(* CODESYS project OC_EtherCAT.library
   DefaultNamespace: OC_EtherCAT
   Description: Open Commissioning TwinCAT EtherCAT Library
   Author: SpiraTec AG
   Title: OC_EtherCAT
   Version: 1.1.8
   Company: Open Commissioning
   Placeholder: OC_EtherCAT

Project tree, tasks and I/O mapping:
  libraries: OC_Core, 1.3.1 (Open Commissioning); OC_TwinSAFE, 1.0.2 (Open Commissioning); Tc2_Math, 3.4.4.0 (Beckhoff Automation GmbH); Tc2_Standard, 3.4.5.0 (Beckhoff Automation GmbH); Tc2_System, 3.6.4.0 (Beckhoff Automation GmbH); Tc3_Module, 3.4.5.0 (Beckhoff Automation GmbH); TcUnit, 1.3.0.0 (www.tcunit.org)
  Devices/
    Drives/
      DS402/
        data type E_DS402_State
        function block FB_DS402_CSP [ST]: Cycle, eState, fbEncoder, GetControlData, InitRun, SetStatusData
        function block FB_DS402_FSM [ST]: bError, eState, IsDisableOperation, IsDisableVoltage, IsEnableOperation, IsFaultReset, IsQuickStop, IsShutdown, IsSwitchOn, nControl, nStatus, ResetError, S0_NotReadyToSwitchOn, S1_SwitchOnDisabled, S2_ReadyToSwitchOn, S3_SwitchedOn, S4_OperationEnabled, S5_Fault, S6_FaultReactionActive, S7_QuickStopActive
        data type ST_DS402_ControlWord
        data type ST_DS402_CSP_Config
        data type ST_DS402_CSP_Control
        data type ST_DS402_CSP_Status
        data type ST_DS402_StatusWord
      Mitsubishi/
        function block FB_Mitsubishi_MRJ4TM [ST]: Cycle, eState, fbEncoder, GetControlData, InitRun, SetStatusData
        data type ST_Mitsubishi_MRJ4TM_Config
        data type ST_Mitsubishi_MRJ4TM_Control
        data type ST_Mitsubishi_MRJ4TM_Status
      Sercos/
        data type E_Sercos_State
        function block FB_Sercos_FSM [ST]: bError, eState, nControl, nStatus, S1_NotReadyToSwitchOn, S2_SwitchOnDisabled, S3_ReadyToSwitchOn, S4_SwitchOn, S5a_DriveInOperation, S5b_Halt, S6_QuickStop, S7_FaultReactionActive, S8_Fault
        function block FB_Sercos_VC [ST]: Cycle, eState, fbEncoder, GetControlData, GetTargetVelocity, InitRun, Motion, SetStatusData
        data type ST_Sercos_ControlWord
        data type ST_Sercos_StatusWord
        data type ST_Sercos_VC
        data type ST_Sercos_VC_Config
        data type ST_Sercos_VC_Control
        data type ST_Sercos_VC_Status
    Terminals/
      FB_Beckhoff_EL6001/
        data type E_Beckhoff_EL6001_State
        function block FB_Beckhoff_EL6001 [ST]: BufferFull, Control, FramingError, InitAccepted, InitRequest, OverrunError, ParityError, ReceiveAccepted, ReceiveRequest, SendContinuous, State, TransmitAccepted, TransmitRequest
      function block FB_Beckhoff_EJ1918 [ST]: FB_init
      function block FB_Beckhoff_EK1914 [ST]: FB_init
      function block FB_Beckhoff_EL1904 [ST]: FB_init
      function block FB_Beckhoff_EL1918 [ST]: FB_init
      function block FB_Beckhoff_EL2904 [ST]: FB_init
      function block FB_Beckhoff_EL5152 [ST]: Control1, Control2, Counter1, Counter2, Period1, Period2, SetCounter1, SetCounter2, Status1, Status2
      function block FB_FSOE_19 [ST]: FB_init
      data type ST_Baumer_Encoder
      data type ST_Beckhoff_16DI
      data type ST_Beckhoff_16DO
      data type ST_Beckhoff_2AI
      data type ST_Beckhoff_4AI
      data type ST_Beckhoff_4AO
      data type ST_Beckhoff_4DI
      data type ST_Beckhoff_4DI_4DO
      data type ST_Beckhoff_4DO
      data type ST_Beckhoff_8DI
      data type ST_Beckhoff_8DI_8DO
      data type ST_Beckhoff_8DO
      data type ST_Beckhoff_EL3403
      data type ST_Beckhoff_EL5002
      data type ST_Beckhoff_EL9110
      data type ST_Beckhoff_EL9410
      data type ST_CoE402
      data type ST_Gefran_GFX4
      data type ST_Mitsubishi_MRJ4TM
      data type ST_SEW_SimMovitrac
*)

// Devices/Drives/DS402/E_DS402_State
{attribute 'qualified_only'}
{attribute 'strict'}
{attribute 'conditionalshow'}
TYPE E_DS402_State :
(
	S0_NotReadyToSwitchOn,
	S1_SwitchOnDisabled,
	S2_ReadyToSwitchOn,
	S3_SwitchedOn,
	S4_OperationEnabled,
	S5_Fault,
	S6_FaultReactionActive,
	S7_QuickStopActive
);
END_TYPE

// Devices/Drives/DS402/ST_DS402_ControlWord
(*
	Object 6040h: Control word (DS402)	
*)
{attribute 'pack_mode' := '0'}
TYPE ST_DS402_ControlWord :
STRUCT
	b0_SwitchOn 					: BIT;
	b1_EnableVoltage				: BIT;
	b2_QuickStop					: BIT;
	b3_EnableOperation				: BIT;
	b4_OperationModeSpecific		: BIT;
	b5_OperationModeSpecific		: BIT;
	b6_OperationModeSpecific		: BIT;
	b7_FaultReset					: BIT;
	b8_Reserved						: BIT;
	b9_Reserved						: BIT;
	b10_Reserved					: BIT;
	b11_Reserved					: BIT;
	b12_Reserved					: BIT;
	b13_Reserved					: BIT;
	b14_Reserved					: BIT;
	b15_Reserved					: BIT;
END_STRUCT
END_TYPE

// Devices/Drives/DS402/ST_DS402_CSP_Config
{attribute 'pack_mode' := '0'}
TYPE ST_DS402_CSP_Config :
STRUCT	
	bForceMode			: BOOL; //Ignore process data from fieldbus.	
	bSwapProcessData	: BOOL; //Reverse process data byte order from/to fieldbus.
	fPositionOffset		: LREAL := 0.0;	
	bSyncOpMode			: BOOL := TRUE;
END_STRUCT
END_TYPE

// Devices/Drives/DS402/ST_DS402_CSP_Control
(*
	Control struct for Cyclic synchronous position mode(CSP)
	0x1600 (DS402 Controlword)
	0x1606 (DS402 Target position)
*)
{attribute 'pack_mode' := '0'}
TYPE ST_DS402_CSP_Control :
STRUCT
	nControlWord 		: ST_DS402_ControlWord; //0x1600 (DS402 Controlword)
	nTargetPosition		: DINT;	//DS402 Target position [INC]	
END_STRUCT
END_TYPE

// Devices/Drives/DS402/ST_DS402_CSP_Status
(*
	Status struct for Cyclic synchronous position mode(CSP)
	0x1A00 (DS402 Statusword)
	0x1A01 (DS402 Position actual value)
	0x1A04 (DS402 Following error actual value)
*)
{attribute 'pack_mode' := '0'}
TYPE ST_DS402_CSP_Status :
STRUCT
	nStatusWord 		: ST_DS402_StatusWord; //0x1A00 (DS402 Statusword)
	nActualPosition		: DINT;	//0x1A01 (DS402 Position actual value) [INC]
	nErrorPosition		: DINT;	//0x1A04 (DS402 Following error actual value) [INC]	
END_STRUCT
END_TYPE

// Devices/Drives/DS402/ST_DS402_StatusWord
(*
	Object 6041h: Status word (DS402)
*)
{attribute 'pack_mode' := '0'}
TYPE ST_DS402_StatusWord :
STRUCT
	b0_ReadyToSwitchOn 				: BIT; 
	b1_SwitchedOn 					: BIT; 
	b2_OperationEnabled 			: BIT; 
	b3_Fault						: BIT; 
	b4_VoltageEnabled				: BIT; 
	b5_QuickStop					: BIT;
	b6_SwitchOnDisabled				: BIT; 
	b7_Warning						: BIT; 
	b8_Synchranisation				: BIT; 
	b9_Remote						: BIT;
	b10_TargetReached				: BIT;
	b11_InternalLimitActive			: BIT; 
	b12_OperationModeSpecific		: BIT; 
	b13_OperationModeSpecific		: BIT; 
	b14_OperationModeSpecific		: BIT; 
	b15_ClosedLoopActive			: BIT;
END_STRUCT
END_TYPE

// Devices/Drives/Mitsubishi/ST_Mitsubishi_MRJ4TM_Config
{attribute 'pack_mode' := '0'}
TYPE ST_Mitsubishi_MRJ4TM_Config :
STRUCT	
	bForceMode			: BOOL; //Ignore process data from fieldbus.	
	bSwapProcessData	: BOOL; //Reverse process data byte order from/to fieldbus.
	fPositionOffset		: LREAL := 0.0;	
	bSyncOpMode			: BOOL := TRUE;
END_STRUCT
END_TYPE

// Devices/Drives/Mitsubishi/ST_Mitsubishi_MRJ4TM_Control
(*
	
*)
{attribute 'pack_mode' := '0'}
TYPE ST_Mitsubishi_MRJ4TM_Control :
STRUCT
	nModesOfOperation 				: SINT;
	nControlWord 					: ST_DS402_ControlWord; //0x1600 (DS402 Controlword)
	nControlID1						: UINT;
	nControlID2						: UINT;
	nControlID3						: UINT;
	nTargetPosit					: DINT;
	nTargetVeloc					: DINT;
	nVelocityLimitValue				: UDINT;
	nTargetTorque					: INT;
	nPositiveTorqueLimitValue		: UINT;
	nNegativeTorqueLimitValue 		: UINT;
	nTouchProbeFunction				: UINT;
END_STRUCT
END_TYPE

// Devices/Drives/Mitsubishi/ST_Mitsubishi_MRJ4TM_Status
(*
	
*)
{attribute 'pack_mode' := '0'}
TYPE ST_Mitsubishi_MRJ4TM_Status :
STRUCT
	nModesOfOperationDisplay 		: SINT;
	nStatusWord 					: ST_DS402_StatusWord; //0x1A00 (DS402 Statusword)
	nStatusDO1						: UINT;
	nStatusDO2						: UINT;
	nStatusDO3						: UINT;
	nPositionActualValue			: DINT;
	nVelocityActualValue			: DINT;
	nFollowingErrorActualValue		: DINT;
	nTorqueActualValue				: INT;
	nTouchProbeStatus				: UINT;
	nTouchProbePos1PosValue			: DINT;
	nTouchProbePos1NegValue			: DINT;
	nTouchProbePos2PosValue			: DINT;
	nTouchProbePos2NegValue			: DINT;
END_STRUCT
END_TYPE

// Devices/Drives/Sercos/E_Sercos_State
{attribute 'qualified_only'}
{attribute 'strict'}
{attribute 'conditionalshow'}
TYPE E_Sercos_State :
(
	S1_NotReadyToSwitchOn,
	S2_SwitchOnDisabled,
	S3_ReadyToSwitchOn,
	S4_SwitchOn,
	S5a_DriveInOperation,
	S5b_Halt,
	S6_QuickStop,
	S7_FaultReactionActive,
	S8_Fault
);
END_TYPE

// Devices/Drives/Sercos/ST_Sercos_ControlWord
(*
	S-0-0134 Drive Control
	https://product-help.schneider-electric.com/Machine%20Expert/V1.2/en/ATV340SUG/ATV340SUG/STI_Software_Setup/STI_Software_Setup-21.htm#XREF_D_SE_0083221_1
*)
{attribute 'pack_mode' := '1'}
TYPE ST_Sercos_ControlWord :
STRUCT
	b0_Reserved 					: BIT;
	b1_Reserved						: BIT;
	b2_Reserved						: BIT;
	b3_Reserved						: BIT;
	b4_Reserved						: BIT;
	b5_Reserved						: BIT;
	b6_Reserved						: BIT;
	b7_Reserved						: BIT;
	b8_Reserved						: BIT; //Reserved (=0)
	b9_Reserved						: BIT; //Reserved (=0)
	b10_OperationMode				: BIT; //0 = Primary operation mode
	b11_Reserved					: BIT;
	b12_Reserved					: BIT; 
	b13_Halt						: BIT; //Drive halt, 1 --> 0 = halt, 0 --> 1 = restart
	b14_Start						: BIT; //Drive start, 1 --> 0 = Stop, 0 -> 1 = Start 
	b15_Enable						: BIT; //Drive enable, 1 --> 0 = drive disabled, 0 -> 1 = drive enabled
END_STRUCT
END_TYPE

// Devices/Drives/Sercos/ST_Sercos_StatusWord
(*
	S-0-0135 Drive Status
	https://product-help.schneider-electric.com/Machine%20Expert/V1.2/en/ATV340SUG/ATV340SUG/STI_Software_Setup/STI_Software_Setup-22.htm#XREF_D_SE_0083227_1
*)
{attribute 'pack_mode' := '1'}
TYPE ST_Sercos_StatusWord :
STRUCT
	b0_Reserved 					: BIT;
	b1_Reserved						: BIT;
	b2_Reserved						: BIT;
	b3_CommandProcessing			: BIT; //Status command value processing if 0 = ignored
	b4_Halt							: BIT; //Drive halt, 0 = inactive, 1 = active
	b5_PositionFeedback				: BIT; //Position feedback value status (S-0-0403)
	b6_Reserved						: BIT;
	b7_QuickStop					: BIT; //Quick stop, 0 = inactive, 1 = active
	b8_Reserved						: BIT; //Reserved (=0)
	b9_Reserved						: BIT; //Reserved (=0)
	b10_OperationMode				: BIT; //0 = Primary operation mode
	b11_Reserved					: BIT;
	b12_Warning						: BIT; //Warning, 0 = No warning, 1 = Warning
	b13_Error						: BIT; //Drive shut-down error, 0 = No error, 1 = Error
	b14_ReadyToOperate				: BIT; //00 = Not ready to switch on, 01 = Switch on disabled, main power disabled
	b15_ReadyToOperate				: BIT; //10 = Switch on, 11 = Drive enabled
END_STRUCT
END_TYPE

// Devices/Drives/Sercos/ST_Sercos_VC
{attribute 'pack_mode' := '1'} 
TYPE ST_Sercos_VC :
STRUCT
	stControl		AT %I* : ST_Sercos_VC_Control;
	stStatus		AT %Q* : ST_Sercos_VC_Status;
END_STRUCT
END_TYPE

// Devices/Drives/Sercos/ST_Sercos_VC_Config
{attribute 'pack_mode' := '0'}
TYPE ST_Sercos_VC_Config :
STRUCT	
	bForceMode				: BOOL; //Ignore process data from fieldbus.	
	bSwapProcessData		: BOOL; //Reverse process data byte order from/to fieldbus.	
	bIsLinkOutputVelocity	: BOOL; //If TRUE, link output is velocity value
	fReferenceVelocity 		: REAL := 1000.0;
	fNormalizationFactor	: REAL := 80000;
END_STRUCT
END_TYPE

// Devices/Drives/Sercos/ST_Sercos_VC_Control
(*
	Sercos Velocity Control
	MDT: S-0-0134 Master control word
	MDT: S-0-0036 Velocity command value
*)
{attribute 'pack_mode' := '0'}
TYPE ST_Sercos_VC_Control :
STRUCT
	nControlWord 			: ST_Sercos_ControlWord; //S-0-0134 Master control word
	nVelocityCommand		: DINT;	//S-0-0036 Velocity command value
END_STRUCT
END_TYPE

// Devices/Drives/Sercos/ST_Sercos_VC_Status
(*
	Sercos Velocity Control
	AT: S-0-0135 Drive Status word
	AT: S-0-0051 Position feedback 1 value
*)
{attribute 'pack_mode' := '0'}
TYPE ST_Sercos_VC_Status :
STRUCT
	nStatusWord 			: ST_Sercos_StatusWord; //S-0-0135 Drive Status word
	nPositionFeedback		: DINT;	//S-0-0051 Position feedback 1 value
END_STRUCT
END_TYPE

// Devices/Terminals/FB_Beckhoff_EL6001/E_Beckhoff_EL6001_State
{attribute 'qualified_only'}
{attribute 'strict'}
TYPE E_Beckhoff_EL6001_State :
(
	INIT,
	READY,
	TRANSMIT, 
	RECEIVE
);
END_TYPE

// Devices/Terminals/ST_Baumer_Encoder
{attribute 'pack_mode' := '1'}
TYPE ST_Baumer_Encoder :
STRUCT
	nPosition		AT %Q*	:	UDINT;
	nWarnings		AT %Q*	:	UINT;
	nSystemTime		AT %Q*	:	UDINT; 
END_STRUCT
END_TYPE

// Devices/Terminals/ST_Beckhoff_16DI
{attribute 'pack_mode' := '1'} 
TYPE ST_Beckhoff_16DI :
STRUCT
	bIn1	AT %Q* : BIT;
	bIn2	AT %Q* : BIT;
	bIn3	AT %Q* : BIT;
	bIn4	AT %Q* : BIT;
	bIn5	AT %Q* : BIT;
	bIn6	AT %Q* : BIT;
	bIn7	AT %Q* : BIT;
	bIn8	AT %Q* : BIT;
	bIn9	AT %Q* : BIT;
	bIn10	AT %Q* : BIT;
	bIn11	AT %Q* : BIT;
	bIn12	AT %Q* : BIT;
	bIn13	AT %Q* : BIT;
	bIn14	AT %Q* : BIT;
	bIn15	AT %Q* : BIT;
	bIn16	AT %Q* : BIT;
END_STRUCT
END_TYPE

// Devices/Terminals/ST_Beckhoff_16DO
{attribute 'pack_mode' := '1'} 
TYPE ST_Beckhoff_16DO :
STRUCT
	bOut1	AT %I* : BIT;
	bOut2	AT %I* : BIT;
	bOut3	AT %I* : BIT;
	bOut4	AT %I* : BIT;
	bOut5	AT %I* : BIT;
	bOut6	AT %I* : BIT;
	bOut7	AT %I* : BIT;
	bOut8	AT %I* : BIT;
	bOut9	AT %I* : BIT;
	bOut10	AT %I* : BIT;
	bOut11	AT %I* : BIT;
	bOut12	AT %I* : BIT;
	bOut13	AT %I* : BIT;
	bOut14	AT %I* : BIT;
	bOut15	AT %I* : BIT;
	bOut16	AT %I* : BIT;
END_STRUCT
END_TYPE

// Devices/Terminals/ST_Beckhoff_2AI
{attribute 'pack_mode' := '1'} 
TYPE ST_Beckhoff_2AI :
STRUCT
	nStatus1	AT %Q* : UINT;
	nValue1		AT %Q* : INT;
	nStatus2	AT %Q* : UINT;
	nValue2		AT %Q* : INT;
	nStatus3	AT %Q* : UINT;
	nValue3		AT %Q* : INT;
	nStatus4	AT %Q* : UINT;
	nValue4		AT %Q* : INT;
END_STRUCT
END_TYPE

// Devices/Terminals/ST_Beckhoff_4AI
{attribute 'pack_mode' := '1'} 
TYPE ST_Beckhoff_4AI :
STRUCT
	nStatus1	AT %Q* : UINT;
	nValue1		AT %Q* : INT;
	nStatus2	AT %Q* : UINT;
	nValue2		AT %Q* : INT;
END_STRUCT
END_TYPE

// Devices/Terminals/ST_Beckhoff_4AO
{attribute 'pack_mode' := '1'} 
TYPE ST_Beckhoff_4AO :
STRUCT
	nAnalogOut1	AT %I* : UINT;
	nAnalogOut2	AT %I* : UINT;
	nAnalogOut3	AT %I* : UINT;
	nAnalogOut4	AT %I* : UINT;
END_STRUCT
END_TYPE

// Devices/Terminals/ST_Beckhoff_4DI
{attribute 'pack_mode' := '1'} 
TYPE ST_Beckhoff_4DI :
STRUCT
	bIn1	AT %Q* : BIT;
	bIn2	AT %Q* : BIT;
	bIn3	AT %Q* : BIT;
	bIn4	AT %Q* : BIT;	
END_STRUCT
END_TYPE

// Devices/Terminals/ST_Beckhoff_4DI_4DO
{attribute 'pack_mode' := '1'} 
TYPE ST_Beckhoff_4DI_4DO :
STRUCT
	bIn1	AT %Q* : BIT;
	bIn2	AT %Q* : BIT;
	bIn3	AT %Q* : BIT;
	bIn4	AT %Q* : BIT;	
	bOut1	AT %I* : BIT;
	bOut2	AT %I* : BIT;
	bOut3	AT %I* : BIT;
	bOut4	AT %I* : BIT;	
END_STRUCT
END_TYPE

// Devices/Terminals/ST_Beckhoff_4DO
{attribute 'pack_mode' := '1'} 
TYPE ST_Beckhoff_4DO :
STRUCT
	bOut1	AT %I* : BIT;
	bOut2	AT %I* : BIT;
	bOut3	AT %I* : BIT;
	bOut4	AT %I* : BIT;	
END_STRUCT
END_TYPE

// Devices/Terminals/ST_Beckhoff_8DI
{attribute 'pack_mode' := '1'} 
TYPE ST_Beckhoff_8DI :
STRUCT
	bIn1	AT %Q* : BIT;
	bIn2	AT %Q* : BIT;
	bIn3	AT %Q* : BIT;
	bIn4	AT %Q* : BIT;
	bIn5	AT %Q* : BIT;
	bIn6	AT %Q* : BIT;
	bIn7	AT %Q* : BIT;
	bIn8	AT %Q* : BIT;
END_STRUCT
END_TYPE

// Devices/Terminals/ST_Beckhoff_8DI_8DO
{attribute 'pack_mode' := '1'} 
TYPE ST_Beckhoff_8DI_8DO :
STRUCT
	bIn1	AT %Q* : BIT;
	bIn2	AT %Q* : BIT;
	bIn3	AT %Q* : BIT;
	bIn4	AT %Q* : BIT;
	bIn5	AT %Q* : BIT;
	bIn6	AT %Q* : BIT;
	bIn7	AT %Q* : BIT;
	bIn8	AT %Q* : BIT;
	bOut1	AT %I* : BIT;
	bOut2	AT %I* : BIT;
	bOut3	AT %I* : BIT;
	bOut4	AT %I* : BIT;
	bOut5	AT %I* : BIT;
	bOut6	AT %I* : BIT;
	bOut7	AT %I* : BIT;
	bOut8	AT %I* : BIT;
END_STRUCT
END_TYPE

// Devices/Terminals/ST_Beckhoff_8DO
{attribute 'pack_mode' := '1'} 
TYPE ST_Beckhoff_8DO :
STRUCT
	bOut1	AT %I* : BIT;
	bOut2	AT %I* : BIT;
	bOut3	AT %I* : BIT;
	bOut4	AT %I* : BIT;
	bOut5	AT %I* : BIT;
	bOut6	AT %I* : BIT;
	bOut7	AT %I* : BIT;
	bOut8	AT %I* : BIT;
END_STRUCT
END_TYPE

// Devices/Terminals/ST_Beckhoff_EL3403
TYPE ST_Beckhoff_EL3403 :
STRUCT
	nCurrent1		AT %Q* : UINT;
	nVoltage1		AT %Q* : UINT;
	nActivePower1	AT %Q* : UINT;
	nCurrent2		AT %Q* : UINT;
	nVoltage2		AT %Q* : UINT;
	nActivePower2	AT %Q* : UINT;	
	nCurrent3		AT %Q* : UINT;
	nVoltage3		AT %Q* : UINT;
	nActivePower3	AT %Q* : UINT;
END_STRUCT
END_TYPE

// Devices/Terminals/ST_Beckhoff_EL5002
TYPE ST_Beckhoff_EL5002 :
STRUCT
	nStatus1	AT %Q* : UINT;
	nCounter1	AT %Q* : UDINT;	
	nStatus2	AT %Q* : UINT;
	nCounter2	AT %Q* : UDINT;	
END_STRUCT
END_TYPE

// Devices/Terminals/ST_Beckhoff_EL9110
{attribute 'pack_mode' := '1'} 
TYPE ST_Beckhoff_EL9110 :
STRUCT
	bPowerOk	AT %Q* : BIT := TRUE;
END_STRUCT
END_TYPE

// Devices/Terminals/ST_Beckhoff_EL9410
{attribute 'pack_mode' := '1'} 
TYPE ST_Beckhoff_EL9410 :
STRUCT
	bUsUndervoltage	AT %Q* : BIT;
	bUpUndervoltage	AT %Q* : BIT;
END_STRUCT
END_TYPE

// Devices/Terminals/ST_CoE402
{attribute 'pack_mode' := '1'} 
TYPE ST_CoE402 :
STRUCT
	nControlWord	AT %I* : UINT;
	nTargetValue	AT %I* : DINT;
	nStatusWord		AT %Q* : UINT;
	nActualValue	AT %Q* : DINT;
END_STRUCT
END_TYPE

// Devices/Terminals/ST_Gefran_GFX4
{attribute 'pack_mode' := '1'} 
TYPE ST_Gefran_GFX4 :
STRUCT
	nProcessVariable1	AT %Q* : INT;
	nControllerStatus1	AT %Q* : UINT;	
	nOutputPower1		AT %Q* : INT;
	nProcessVariable2	AT %Q* : INT;
	nControllerStatus2	AT %Q* : UINT;	
	nOutputPower2		AT %Q* : INT;
	nProcessVariable3	AT %Q* : INT;
	nControllerStatus3	AT %Q* : UINT;	
	nOutputPower3		AT %Q* : INT;
	nProcessVariable4	AT %Q* : INT;
	nControllerStatus4	AT %Q* : UINT;	
	nOutputPower4		AT %Q* : INT;
	nLocalSetpoint1		AT %I* : INT;
	nLocalSetpoint2		AT %I* : INT;
	nLocalSetpoint3		AT %I* : INT;
	nLocalSetpoint4		AT %I* : INT;
END_STRUCT
END_TYPE

// Devices/Terminals/ST_Mitsubishi_MRJ4TM
{attribute 'pack_mode' := '1'} 
TYPE ST_Mitsubishi_MRJ4TM :
STRUCT
	nModesOfOperation 				AT %I* : SINT;
	nControlWord					AT %I* : UINT;
	nControlID1						AT %I* : UINT;
	nControlID2						AT %I* : UINT;
	nControlID3						AT %I* : UINT;
	nTargetPosit					AT %I* : DINT;
	nTargetVeloc					AT %I* : DINT;
	nVelocityLimitValue				AT %I* : UDINT;
	nTargetTorque					AT %I* : INT;
	nPositiveTorqueLimitValue		AT %I* : UINT;
	nNegativeTorqueLimitValue 		AT %I* : UINT;
	nTouchProbeFunction				AT %I* : UINT;
	
	nModesOfOperationDisplay 		AT %Q* : SINT;
	nStatusWord						AT %Q* : UINT;
	nStatusDO1						AT %Q* : UINT;
	nStatusDO2						AT %Q* : UINT;
	nStatusDO3						AT %Q* : UINT;
	nPositionActualValue			AT %Q* : DINT;
	nVelocityActualValue			AT %Q* : DINT;
	nFollowingErrorActualValue		AT %Q* : DINT;
	nTorqueActualValue				AT %Q* : INT;
	nTouchProbeStatus				AT %Q* : UINT;
	nTouchProbePos1PosValue			AT %Q* : DINT;
	nTouchProbePos1NegValue			AT %Q* : DINT;
	nTouchProbePos2PosValue			AT %Q* : DINT;
	nTouchProbePos2NegValue			AT %Q* : DINT;
END_STRUCT
END_TYPE

// Devices/Terminals/ST_SEW_SimMovitrac
{attribute 'pack_mode' := '1'}
TYPE ST_SEW_SimMovitrac :
STRUCT
	PI1		AT %Q* : WORD;
	PI2		AT %Q* : WORD;
	PI3		AT %Q* : WORD;
	PO1		AT %I* : WORD;
	PO2		AT %I* : WORD;
	PO3		AT %I* : WORD;
END_STRUCT
END_TYPE

// Devices/Drives/DS402/FB_DS402_CSP
(*
	DS402 with Cyclic synchronous position mode(CSP)
	SM2 PDO: 0x1600 (DS402 Controlword)	
	SM2 PDO: 0x1606 (DS402 Target position)
	SM3 PDO: 0x1A00 (DS402 Statusword)	
	SM3 PDO: 0x1A01 (DS402 Position actual value)
	SM3 PDO: 0x1A04 (DS402 Following error actual value)
*)
{attribute 'reflection'} 
FUNCTION_BLOCK FB_DS402_CSP EXTENDS FB_LinkDataReal 
VAR_INPUT
	pControl			: PVOID; //Pocess data from fieldbus, 6 BYTES FROM FIELDBUS
	pStatus				: PVOID; //Pocess data to fieldbus, 6 BYTES FROM FIELDBUS		
	stControl	 		: ST_DS402_CSP_Control;
	stConfig			: ST_DS402_CSP_Config;
	bSTO 				: BOOL := TRUE;
END_VAR

VAR_OUTPUT
	stStatus 			: ST_DS402_CSP_Status;	
END_VAR

VAR		
	{attribute 'instance-path'} 
    {attribute 'noinit'} 
    _sPath 				: STRING;
	_fbStateMachine 	: FB_DS402_FSM;
	_fbEncoder 			: FB_Encoder;	
END_VAR

SUPER^();
InitRun();

GetControlData();
Cycle();
SetStatusData();

METHOD PRIVATE Cycle
IF NOT bSTO THEN RETURN; END_IF

_fbStateMachine.stControl := stControl.nControlWord;
_fbStateMachine();
stStatus.nStatusWord := _fbStateMachine.stStatus;

IF (_fbStateMachine._eState = E_DS402_State.S4_OperationEnabled) THEN	
	
	_fbEncoder.fValue :=  stConfig.fPositionOffset + _fbEncoder.INC_TO_LREAL(stControl.nTargetPosition, 1);
	_fbEncoder();
END_IF

IF stConfig.bSyncOpMode THEN
	stStatus.nStatusWord.b12_OperationModeSpecific := stControl.nControlWord.b4_OperationModeSpecific;
	stStatus.nStatusWord.b13_OperationModeSpecific := stControl.nControlWord.b5_OperationModeSpecific;
	stStatus.nStatusWord.b14_OperationModeSpecific := stControl.nControlWord.b6_OperationModeSpecific;
END_IF


stStatus.nActualPosition := _fbEncoder.nResult;

//Set Link Data
ControlData := LREAL_TO_REAL(_fbEncoder.fResult);
END_METHOD

PROPERTY eState : E_DS402_State
GET
eState := _fbStateMachine.eState;
END_GET
END_PROPERTY

PROPERTY PUBLIC fbEncoder : REFERENCE TO FB_Encoder
GET
fbEncoder REF= _fbEncoder;
END_GET
END_PROPERTY

METHOD INTERNAL GetControlData
IF pControl <= 0 OR stConfig.bForceMode THEN RETURN; END_IF

(*Control Word*)
F_Memcpy(ADR(stControl), pControl, 2, stConfig.bSwapProcessData);
(*Target Value*)
F_Memcpy(ADR(stControl) + 2, pControl + 2, 4, stConfig.bSwapProcessData);
END_METHOD

METHOD PRIVATE InitRun
VAR_INST
	bInitRun : BOOL := TRUE;
END_VAR
IF NOT bInitRun THEN RETURN; END_IF
bInitRun := FALSE;

IF pControl = 0 OR pStatus = 0 THEN
	ADSLOGSTR(ADSLOG_MSGTYPE_WARN, '%s', CONCAT(_sPath, ' PLC IO is not assigned!'));	
END_IF
END_METHOD

METHOD INTERNAL SetStatusData
IF pStatus <= 0 THEN RETURN; END_IF

(*StatusWord*)
F_Memcpy(pStatus, ADR(stStatus), 2, stConfig.bSwapProcessData);
(*Actual Position*)
F_Memcpy(pStatus + 2, ADR(stStatus) + 2, 4, stConfig.bSwapProcessData);
(*Actual Position Error*)
F_Memcpy(pStatus + 6, ADR(stStatus) + 6, 4, stConfig.bSwapProcessData);
END_METHOD

END_FUNCTION_BLOCK

// Devices/Drives/DS402/FB_DS402_FSM
(*
	DS402 Finite State Machine General
*)
FUNCTION_BLOCK FB_DS402_FSM
VAR_INPUT	
	stControl					: ST_DS402_ControlWord;
END_VAR

VAR_OUTPUT	
	stStatus					: ST_DS402_StatusWord;	
END_VAR

VAR	
	_eState 					: E_DS402_State := E_DS402_State.S0_NotReadyToSwitchOn;	
	_rTrig_QuickStop 			: R_TRIG;
	_rTrig_Reset 				: R_TRIG;
	_bError						: BOOL;
END_VAR

_rTrig_QuickStop(CLK := stControl.b2_QuickStop);
_rTrig_Reset(CLK := stControl.b7_FaultReset);

CASE _eState OF
	E_DS402_State.S0_NotReadyToSwitchOn : S0_NotReadyToSwitchOn();
	E_DS402_State.S1_SwitchOnDisabled : S1_SwitchOnDisabled();
	E_DS402_State.S2_ReadyToSwitchOn : S2_ReadyToSwitchOn();
	E_DS402_State.S3_SwitchedOn : S3_SwitchedOn();
	E_DS402_State.S4_OperationEnabled : S4_OperationEnabled();
	E_DS402_State.S5_Fault : S5_Fault();	
	E_DS402_State.S6_FaultReactionActive : S6_FaultReactionActive();	
	E_DS402_State.S7_QuickStopActive : S7_QuickStopActive();			
END_CASE

PROPERTY PUBLIC bError : BOOL
GET
bError := _bError;
END_GET
SET
IF bError AND NOT _bError THEN
	_bError := TRUE;
END_IF
END_SET
END_PROPERTY

PROPERTY eState : E_DS402_State
GET
eState := _eState;
END_GET
SET
_eState := eState;
END_SET
END_PROPERTY

METHOD PRIVATE IsDisableOperation : BOOL
IsDisableOperation := 
stControl.b0_SwitchOn 
AND stControl.b1_EnableVoltage 
AND stControl.b2_QuickStop 
AND NOT stControl.b3_EnableOperation
AND NOT stControl.b7_FaultReset;
END_METHOD

METHOD PRIVATE IsDisableVoltage : BOOL
IsDisableVoltage := 
NOT stControl.b1_EnableVoltage
AND NOT stControl.b7_FaultReset;
END_METHOD

METHOD PRIVATE IsEnableOperation : BOOL
IsEnableOperation := 
stControl.b0_SwitchOn 
AND stControl.b1_EnableVoltage 
AND stControl.b2_QuickStop 
AND stControl.b3_EnableOperation
AND NOT stControl.b7_FaultReset;
END_METHOD

METHOD PRIVATE IsFaultReset : BOOL
IsFaultReset := _rTrig_Reset.Q;
END_METHOD

METHOD PRIVATE IsQuickStop : BOOL
IsQuickStop := 
NOT stControl.b2_QuickStop
AND NOT stControl.b7_FaultReset;
END_METHOD

METHOD PRIVATE IsShutdown : BOOL
IsShutdown := 
NOT stControl.b0_SwitchOn 
AND stControl.b1_EnableVoltage 
AND stControl.b2_QuickStop
AND NOT stControl.b7_FaultReset;
END_METHOD

METHOD PRIVATE IsSwitchOn : BOOL
IsSwitchOn := 
stControl.b0_SwitchOn 
AND stControl.b1_EnableVoltage 
AND stControl.b2_QuickStop
AND NOT stControl.b7_FaultReset;
END_METHOD

PROPERTY nControl : WORD
GET
nControl.0	:= stControl.b0_SwitchOn;					         
nControl.1	:= stControl.b1_EnableVoltage;				      	
nControl.2	:= stControl.b2_QuickStop;					         	
nControl.3	:= stControl.b3_EnableOperation;			     	
nControl.4	:= stControl.b4_OperationModeSpecific;			
nControl.5	:= stControl.b5_OperationModeSpecific;			
nControl.6	:= stControl.b6_OperationModeSpecific;			
nControl.7	:= stControl.b7_FaultReset;					        	
nControl.8	:= stControl.b8_Reserved;					          	
nControl.9	:= stControl.b9_Reserved;					          
nControl.10	:= stControl.b10_Reserved;					         	
nControl.11	:= stControl.b11_Reserved;					         	
nControl.12	:= stControl.b12_Reserved;					         	
nControl.13	:= stControl.b13_Reserved;					         	
nControl.14	:= stControl.b14_Reserved;					         	
nControl.15 := stControl.b15_Reserved;
END_GET
SET
stControl.b0_SwitchOn 					:= 	nControl.0;	
stControl.b1_EnableVoltage				:= 	nControl.1;		
stControl.b2_QuickStop					:= 	nControl.2;		
stControl.b3_EnableOperation			:= 	nControl.3;		
stControl.b4_OperationModeSpecific		:= 	nControl.4;		
stControl.b5_OperationModeSpecific		:= 	nControl.5;		
stControl.b6_OperationModeSpecific		:= 	nControl.6;		
stControl.b7_FaultReset					:= 	nControl.7;		
stControl.b8_Reserved					:= 	nControl.8;		
stControl.b9_Reserved					:= 	nControl.9;		
stControl.b10_Reserved					:= 	nControl.10;		
stControl.b11_Reserved					:= 	nControl.11;		
stControl.b12_Reserved					:= 	nControl.12;		
stControl.b13_Reserved					:= 	nControl.13;		
stControl.b14_Reserved					:= 	nControl.14;		
stControl.b15_Reserved					:= 	nControl.15;
END_SET
END_PROPERTY

PROPERTY nStatus : WORD
GET
nStatus.0 := stStatus.b0_ReadyToSwitchOn; 			
nStatus.1 := stStatus.b1_SwitchedOn; 				
nStatus.2 := stStatus.b2_OperationEnabled;			
nStatus.3 := stStatus.b3_Fault;					
nStatus.4 := stStatus.b4_VoltageEnabled;
nStatus.5 := stStatus.b5_QuickStop;
nStatus.6 := stStatus.b6_SwitchOnDisabled;			
nStatus.7 := stStatus.b7_Warning;					
nStatus.8 := stStatus.b8_Synchranisation;			
nStatus.9 := stStatus.b9_Remote;			
nStatus.10 := stStatus.b10_TargetReached;				
nStatus.11 := stStatus.b11_InternalLimitActive;		
nStatus.12 := stStatus.b12_OperationModeSpecific;			
nStatus.13 := stStatus.b13_OperationModeSpecific;			
nStatus.14 := stStatus.b14_OperationModeSpecific;			
nStatus.15 := stStatus.b15_ClosedLoopActive;
END_GET
END_PROPERTY

METHOD INTERNAL ResetError : BOOL
_bError := FALSE;
END_METHOD

METHOD PRIVATE S0_NotReadyToSwitchOn : BOOL
VAR_INPUT
END_VAR
stStatus.b0_ReadyToSwitchOn 		:= FALSE;
stStatus.b1_SwitchedOn 				:= FALSE;
stStatus.b2_OperationEnabled		:= FALSE;
stStatus.b3_Fault					:= FALSE;
stStatus.b4_VoltageEnabled			:= FALSE;
stStatus.b6_SwitchOnDisabled 		:= FALSE;

_eState := E_DS402_State.S1_SwitchOnDisabled;
END_METHOD

METHOD PRIVATE S1_SwitchOnDisabled : BOOL
VAR_INPUT
END_VAR
stStatus.b0_ReadyToSwitchOn 		:= FALSE;
stStatus.b1_SwitchedOn				:= FALSE;
stStatus.b2_OperationEnabled 		:= FALSE;
stStatus.b3_Fault 					:= FALSE;
stStatus.b4_VoltageEnabled			:= FALSE;
stStatus.b6_SwitchOnDisabled 		:= TRUE;

IF IsShutdown() THEN
	_eState := E_DS402_State.S2_ReadyToSwitchOn;
END_IF
END_METHOD

METHOD PRIVATE S2_ReadyToSwitchOn : BOOL
VAR_INPUT
END_VAR
stStatus.b0_ReadyToSwitchOn 		:= TRUE;
stStatus.b1_SwitchedOn 				:= FALSE;
stStatus.b2_OperationEnabled 		:= FALSE;
stStatus.b3_Fault 					:= FALSE;
stStatus.b4_VoltageEnabled			:= TRUE;
stStatus.b5_QuickStop 				:= TRUE; 
stStatus.b6_SwitchOnDisabled 		:= FALSE;

IF _bError THEN
	_eState := E_DS402_State.S6_FaultReactionActive;
	RETURN;
END_IF

IF IsDisableVoltage() OR IsQuickStop() THEN
	_eState := E_DS402_State.S1_SwitchOnDisabled;
	RETURN;
END_IF

IF IsSwitchOn() THEN
	_eState := E_DS402_State.S3_SwitchedOn;
	RETURN;
END_IF
END_METHOD

METHOD PRIVATE S3_SwitchedOn : BOOL
VAR_INPUT
END_VAR
stStatus.b0_ReadyToSwitchOn 		:= TRUE;
stStatus.b1_SwitchedOn 				:= TRUE;
stStatus.b2_OperationEnabled 		:= FALSE;
stStatus.b3_Fault 					:= FALSE;
stStatus.b5_QuickStop 				:= TRUE; 
stStatus.b6_SwitchOnDisabled 		:= FALSE;

IF _bError THEN
	_eState := E_DS402_State.S6_FaultReactionActive;
	RETURN;
END_IF

IF IsDisableVoltage() OR IsQuickStop() THEN
	_eState := E_DS402_State.S1_SwitchOnDisabled;
	RETURN;
END_IF

IF IsShutdown() THEN
	_eState := E_DS402_State.S2_ReadyToSwitchOn;
	RETURN;
END_IF

IF IsEnableOperation() THEN
	_eState := E_DS402_State.S4_OperationEnabled;
	RETURN;
END_IF
END_METHOD

METHOD PRIVATE S4_OperationEnabled : BOOL
VAR_INPUT
END_VAR
stStatus.b0_ReadyToSwitchOn				:= TRUE;
stStatus.b1_SwitchedOn 					:= TRUE;
stStatus.b2_OperationEnabled 			:= TRUE;
stStatus.b3_Fault 						:= FALSE;
stStatus.b5_QuickStop 					:= TRUE; 
stStatus.b6_SwitchOnDisabled 			:= FALSE;

IF _bError THEN
	_eState := E_DS402_State.S6_FaultReactionActive;
	RETURN;
END_IF

IF IsDisableVoltage() THEN
	_eState := E_DS402_State.S1_SwitchOnDisabled;
	RETURN;
END_IF

IF IsShutdown() THEN
	_eState := E_DS402_State.S2_ReadyToSwitchOn;
	RETURN;
END_IF

IF IsQuickStop() THEN
	_eState := E_DS402_State.S7_QuickStopActive;
	RETURN;
END_IF

IF IsDisableOperation() THEN
	_eState := E_DS402_State.S3_SwitchedOn;
	RETURN;
END_IF
END_METHOD

METHOD PRIVATE S5_Fault : BOOL
VAR_INPUT
END_VAR
stStatus.b0_ReadyToSwitchOn 		:= FALSE;
stStatus.b1_SwitchedOn				:= FALSE;
stStatus.b2_OperationEnabled 		:= FALSE;
stStatus.b3_Fault 					:= TRUE;
stStatus.b6_SwitchOnDisabled 		:= FALSE;

IF IsFaultReset() THEN
	_bError := FALSE;
	_eState := E_DS402_State.S1_SwitchOnDisabled;
	RETURN;
END_IF
END_METHOD

METHOD PRIVATE S6_FaultReactionActive : BOOL
VAR_INPUT
END_VAR
stStatus.b0_ReadyToSwitchOn 		:= TRUE;
stStatus.b1_SwitchedOn 				:= TRUE;
stStatus.b2_OperationEnabled 		:= TRUE;
stStatus.b3_Fault 					:= TRUE;
stStatus.b6_SwitchOnDisabled 		:= FALSE;

_eState := E_DS402_State.S5_Fault;
END_METHOD

METHOD PRIVATE S7_QuickStopActive : BOOL
VAR_INPUT
END_VAR
stStatus.b0_ReadyToSwitchOn 		:= TRUE;
stStatus.b1_SwitchedOn 				:= TRUE;
stStatus.b2_OperationEnabled 		:= TRUE;
stStatus.b3_Fault 					:= FALSE;
stStatus.b5_QuickStop 				:= FALSE; 
stStatus.b6_SwitchOnDisabled		:= FALSE;

IF IsDisableVoltage() THEN
	_eState := E_DS402_State.S1_SwitchOnDisabled;
	RETURN;
END_IF

IF IsEnableOperation() THEN
	_eState := E_DS402_State.S4_OperationEnabled;
	RETURN;
END_IF
END_METHOD

END_FUNCTION_BLOCK

// Devices/Drives/Mitsubishi/FB_Mitsubishi_MRJ4TM
(*
	
*)
{attribute 'reflection'} 
FUNCTION_BLOCK FB_Mitsubishi_MRJ4TM EXTENDS FB_LinkDataReal 
VAR_INPUT
	pControl			: PVOID; //Pocess data from fieldbus, 29 BYTES FROM FIELDBUS
	pStatus				: PVOID; //Pocess data to fieldbus, 41 BYTES FROM FIELDBUS		
	stControl	 		: ST_Mitsubishi_MRJ4TM_Control;
	stConfig			: ST_Mitsubishi_MRJ4TM_Config;
	bSTO 				: BOOL := TRUE;
END_VAR

VAR_OUTPUT
	stStatus 			: ST_Mitsubishi_MRJ4TM_Status;	
END_VAR

VAR		
	{attribute 'instance-path'} 
    {attribute 'noinit'} 
    _sPath 				: STRING;
	_fbStateMachine 	: FB_DS402_FSM;
	_fbEncoder 			: FB_Encoder;	
END_VAR

SUPER^();
InitRun();

GetControlData();
Cycle();
SetStatusData();

METHOD PRIVATE Cycle
IF NOT bSTO THEN RETURN; END_IF

_fbStateMachine.stControl := stControl.nControlWord;
_fbStateMachine();
stStatus.nStatusWord := _fbStateMachine.stStatus;

IF (_fbStateMachine._eState = E_DS402_State.S4_OperationEnabled) THEN	
	
	_fbEncoder.fValue :=  stConfig.fPositionOffset + _fbEncoder.INC_TO_LREAL(stControl.nTargetPosit, 1);
	_fbEncoder();
END_IF

IF stConfig.bSyncOpMode THEN
	stStatus.nStatusWord.b12_OperationModeSpecific := stControl.nControlWord.b4_OperationModeSpecific;
	stStatus.nStatusWord.b13_OperationModeSpecific := stControl.nControlWord.b5_OperationModeSpecific;
	stStatus.nStatusWord.b14_OperationModeSpecific := stControl.nControlWord.b6_OperationModeSpecific;
END_IF


stStatus.nPositionActualValue := _fbEncoder.nResult;
stStatus.nModesOfOperationDisplay := stControl.nModesOfOperation;

//Set Link Data
ControlData := LREAL_TO_REAL(_fbEncoder.fResult);
END_METHOD

PROPERTY eState : E_DS402_State
GET
eState := _fbStateMachine.eState;
END_GET
END_PROPERTY

PROPERTY PUBLIC fbEncoder : REFERENCE TO FB_Encoder
GET
fbEncoder REF= _fbEncoder;
END_GET
END_PROPERTY

METHOD INTERNAL GetControlData
IF pControl <= 0 OR stConfig.bForceMode THEN RETURN; END_IF

(*nModesOfOperation*) 			F_Memcpy(ADR(stControl), pControl, 1, stConfig.bSwapProcessData);
(*nControlWord*)				F_Memcpy(ADR(stControl)+ 1, pControl + 1, 2, stConfig.bSwapProcessData);
(*nControlID1*)					F_Memcpy(ADR(stControl) + 3, pControl + 3, 2, stConfig.bSwapProcessData);
(*nControlID2*)					F_Memcpy(ADR(stControl) + 5, pControl + 5, 2, stConfig.bSwapProcessData);
(*nControlID3*)					F_Memcpy(ADR(stControl) + 7, pControl + 7, 2, stConfig.bSwapProcessData);
(*nTargetPosit*)				F_Memcpy(ADR(stControl) + 9, pControl + 9, 4, stConfig.bSwapProcessData);
(*nTargetVeloc*)				F_Memcpy(ADR(stControl) + 13, pControl + 13, 4, stConfig.bSwapProcessData);
(*nVelocityLimitValue*)			F_Memcpy(ADR(stControl) + 17, pControl + 17, 4, stConfig.bSwapProcessData);
(*nTargetTorque*)				F_Memcpy(ADR(stControl) + 21, pControl + 21, 2, stConfig.bSwapProcessData);
(*nPositiveTorqueLimitValue*)	F_Memcpy(ADR(stControl) + 23, pControl + 23, 2, stConfig.bSwapProcessData);
(*nNegativeTorqueLimitValue*)	F_Memcpy(ADR(stControl) + 25, pControl + 25, 2, stConfig.bSwapProcessData);
(*nTouchProbeFunction*)			F_Memcpy(ADR(stControl) + 27, pControl + 27, 2, stConfig.bSwapProcessData);
END_METHOD

METHOD PRIVATE InitRun
VAR_INST
	bInitRun : BOOL := TRUE;
END_VAR
IF NOT bInitRun THEN RETURN; END_IF
bInitRun := FALSE;

IF pControl = 0 OR pStatus = 0 THEN
	ADSLOGSTR(ADSLOG_MSGTYPE_WARN, '%s', CONCAT(_sPath, ' PLC IO is not assigned!'));	
END_IF
END_METHOD

METHOD INTERNAL SetStatusData
IF pStatus <= 0 THEN RETURN; END_IF

(*nModesOfOperationDisplay*) 	F_Memcpy(pStatus, ADR(stStatus), 1, stConfig.bSwapProcessData);
(*nStatusWord*) 				F_Memcpy(pStatus + 1, ADR(stStatus) + 1, 2, stConfig.bSwapProcessData);
(*nStatusDO1*) 					F_Memcpy(pStatus + 3, ADR(stStatus) + 3, 2, stConfig.bSwapProcessData);
(*nStatusDO2*) 					F_Memcpy(pStatus + 5, ADR(stStatus) + 5, 2, stConfig.bSwapProcessData);
(*nStatusDO3*) 					F_Memcpy(pStatus + 7, ADR(stStatus) + 7, 2, stConfig.bSwapProcessData);
(*nPositionActualValue*) 		F_Memcpy(pStatus + 9, ADR(stStatus) + 9, 4, stConfig.bSwapProcessData);
(*nVelocityActualValue*) 		F_Memcpy(pStatus + 13, ADR(stStatus) + 13, 4, stConfig.bSwapProcessData);
(*nFollowingErrorActualValue*) 	F_Memcpy(pStatus + 17, ADR(stStatus) + 17, 4, stConfig.bSwapProcessData);
(*nTorqueActualValue*) 			F_Memcpy(pStatus + 21, ADR(stStatus) + 21, 2, stConfig.bSwapProcessData);
(*nTouchProbeStatus*) 			F_Memcpy(pStatus + 23, ADR(stStatus) + 23, 2, stConfig.bSwapProcessData);
(*nTouchProbePos1PosValue*) 	F_Memcpy(pStatus + 25, ADR(stStatus) + 25, 4, stConfig.bSwapProcessData);
(*nTouchProbePos1NegValue*) 	F_Memcpy(pStatus + 29, ADR(stStatus) + 29, 4, stConfig.bSwapProcessData);
(*nTouchProbePos2PosValue*) 	F_Memcpy(pStatus + 33, ADR(stStatus) + 33, 4, stConfig.bSwapProcessData);
(*nTouchProbePos2NegValue*) 	F_Memcpy(pStatus + 37, ADR(stStatus) + 37, 4, stConfig.bSwapProcessData);
END_METHOD

END_FUNCTION_BLOCK

// Devices/Drives/Sercos/FB_Sercos_FSM
(*
	Sercos Finite State Machine General
*)
FUNCTION_BLOCK FB_Sercos_FSM
VAR_INPUT
	bPower						: BOOL := TRUE;	
	stControl					: ST_Sercos_ControlWord;
END_VAR

VAR_OUTPUT	
	stStatus					: ST_Sercos_StatusWord;	
END_VAR

VAR	
	_eState 					: E_Sercos_State := E_Sercos_State.S1_NotReadyToSwitchOn;
	_rTrig_Reset 				: R_TRIG;
	_bError						: BOOL;
END_VAR

_rTrig_Reset(CLK := stControl.b13_Halt);

CASE _eState OF
	E_Sercos_State.S1_NotReadyToSwitchOn 	: S1_NotReadyToSwitchOn();
	E_Sercos_State.S2_SwitchOnDisabled 		: S2_SwitchOnDisabled();
	E_Sercos_State.S3_ReadyToSwitchOn 		: S3_ReadyToSwitchOn();
	E_Sercos_State.S4_SwitchOn 				: S4_SwitchOn();
	E_Sercos_State.S5a_DriveInOperation 	: S5a_DriveInOperation();
	E_Sercos_State.S5b_Halt 				: S5b_Halt();	
	E_Sercos_State.S6_QuickStop 			: S6_QuickStop();	
	E_Sercos_State.S7_FaultReactionActive 	: S7_FaultReactionActive();
	E_Sercos_State.S8_Fault 				: S8_Fault();
END_CASE

PROPERTY PUBLIC bError : BOOL
GET
bError := _bError;
END_GET
SET
_bError := bError;
END_SET
END_PROPERTY

PROPERTY eState : E_Sercos_State
GET
eState := _eState;
END_GET
SET
_eState := eState;
END_SET
END_PROPERTY

PROPERTY nControl : WORD
GET
nControl.0	:= stControl.b0_Reserved;					           
nControl.1	:= stControl.b1_Reserved;						        	
nControl.2	:= stControl.b2_Reserved;						           	
nControl.3	:= stControl.b3_Reserved;						       	
nControl.4	:= stControl.b4_Reserved;						    
nControl.5	:= stControl.b5_Reserved;						    
nControl.6	:= stControl.b6_Reserved;						    
nControl.7	:= stControl.b7_Reserved;						          	
nControl.8	:= stControl.b8_Reserved;						            	
nControl.9	:= stControl.b9_Reserved;						            
nControl.10	:= stControl.b10_OperationMode;				       	
nControl.11	:= stControl.b11_Reserved;					           	
nControl.12	:= stControl.b12_Reserved;
nControl.13	:= stControl.b13_Halt;						              	
nControl.14	:= stControl.b14_Start;						            	
nControl.15 := stControl.b15_Enable;
END_GET
SET
stControl.b0_Reserved 					:= 	nControl.0;	
stControl.b1_Reserved					:= 	nControl.1;		
stControl.b2_Reserved					:= 	nControl.2;		
stControl.b3_Reserved					:= 	nControl.3;		
stControl.b4_Reserved					:= 	nControl.4;		
stControl.b5_Reserved					:= 	nControl.5;		
stControl.b6_Reserved					:= 	nControl.6;		
stControl.b7_Reserved					:= 	nControl.7;		
stControl.b8_Reserved					:= 	nControl.8;		
stControl.b9_Reserved					:= 	nControl.9;		
stControl.b10_OperationMode				:= 	nControl.10;		
stControl.b11_Reserved					:= 	nControl.11;		
stControl.b12_Reserved					:= 	nControl.12;		
stControl.b13_Halt						:= 	nControl.13;		
stControl.b14_Start					:= 	nControl.14;		
stControl.b15_Enable						:= 	nControl.15;
END_SET
END_PROPERTY

PROPERTY nStatus : WORD
GET
nStatus.0 	:= stStatus.b0_Reserved;					      
nStatus.1 	:= stStatus.b1_Reserved;						      
nStatus.2 	:= stStatus.b2_Reserved;						      
nStatus.3 	:= stStatus.b3_CommandProcessing;		
nStatus.4 	:= stStatus.b4_Halt;							         
nStatus.5 	:= stStatus.b5_PositionFeedback;		
nStatus.6 	:= stStatus.b6_Reserved;					      
nStatus.7 	:= stStatus.b7_QuickStop;					      
nStatus.8 	:= stStatus.b8_Reserved;					      
nStatus.9 	:= stStatus.b9_Reserved;					      
nStatus.10 	:= stStatus.b10_OperationMode;		  
nStatus.11 	:= stStatus.b11_Reserved;					      
nStatus.12 	:= stStatus.b12_Warning;					      
nStatus.13 	:= stStatus.b13_Error;					        
nStatus.14 	:= stStatus.b14_ReadyToOperate;			 
nStatus.15 	:= stStatus.b15_ReadyToOperate;
END_GET
END_PROPERTY

METHOD PRIVATE S1_NotReadyToSwitchOn : BOOL
VAR_INPUT
END_VAR
stStatus.b15_ReadyToOperate 		:= FALSE;
stStatus.b14_ReadyToOperate 		:= FALSE;
stStatus.b13_Error 					:= FALSE;
stStatus.b7_QuickStop 				:= FALSE;
stStatus.b4_Halt 					:= FALSE;
stStatus.b3_CommandProcessing 		:= FALSE;

_eState := E_Sercos_State.S2_SwitchOnDisabled;
END_METHOD

METHOD PRIVATE S2_SwitchOnDisabled : BOOL
VAR_INPUT
END_VAR
stStatus.b15_ReadyToOperate 		:= FALSE;
stStatus.b14_ReadyToOperate 		:= TRUE;
stStatus.b13_Error 					:= FALSE;
stStatus.b7_QuickStop 				:= FALSE;
stStatus.b4_Halt 					:= FALSE;
stStatus.b3_CommandProcessing 		:= FALSE;

IF bPower THEN
	_eState := E_Sercos_State.S3_ReadyToSwitchOn;
	RETURN;
END_IF
END_METHOD

METHOD PRIVATE S3_ReadyToSwitchOn : BOOL
VAR_INPUT
END_VAR
stStatus.b15_ReadyToOperate 		:= TRUE;
stStatus.b14_ReadyToOperate 		:= FALSE;
stStatus.b13_Error 					:= FALSE;
stStatus.b7_QuickStop 				:= FALSE;
stStatus.b4_Halt 					:= FALSE;
stStatus.b3_CommandProcessing 		:= FALSE;

IF NOT bPower THEN
	_eState := E_Sercos_State.S2_SwitchOnDisabled;
	RETURN;
END_IF

IF _bError THEN
	_eState := E_Sercos_State.S7_FaultReactionActive;
	RETURN;
END_IF

IF stControl.b15_Enable THEN
	_eState := E_Sercos_State.S4_SwitchOn;
	RETURN;
END_IF
END_METHOD

METHOD PRIVATE S4_SwitchOn : BOOL
VAR_INPUT
END_VAR
stStatus.b15_ReadyToOperate 		:= FALSE;
stStatus.b14_ReadyToOperate 		:= TRUE;
stStatus.b13_Error 					:= FALSE;
stStatus.b7_QuickStop 				:= FALSE;
stStatus.b4_Halt 					:= FALSE;
stStatus.b3_CommandProcessing 		:= FALSE;

IF NOT bPower THEN
	_eState := E_Sercos_State.S2_SwitchOnDisabled;
	RETURN;
END_IF

IF _bError THEN
	_eState := E_Sercos_State.S7_FaultReactionActive;
	RETURN;
END_IF

IF NOT stControl.b15_Enable THEN 
	_eState := E_Sercos_State.S3_ReadyToSwitchOn;
	RETURN;
END_IF

IF stControl.b13_Halt AND stControl.b14_Start THEN
	_eState := E_Sercos_State.S5b_Halt;
	RETURN;
END_IF

IF NOT stControl.b13_Halt AND stControl.b14_Start THEN
	_eState := E_Sercos_State.S5a_DriveInOperation;
	RETURN;
END_IF
END_METHOD

METHOD PRIVATE S5a_DriveInOperation : BOOL
VAR_INPUT
END_VAR
stStatus.b15_ReadyToOperate 		:= TRUE;
stStatus.b14_ReadyToOperate 		:= TRUE;
stStatus.b13_Error 					:= FALSE;
stStatus.b7_QuickStop 				:= FALSE;
stStatus.b4_Halt 					:= FALSE;
stStatus.b3_CommandProcessing 		:= TRUE;

IF NOT bPower THEN
	_eState := E_Sercos_State.S2_SwitchOnDisabled;
	RETURN;
END_IF

IF _bError THEN
	_eState := E_Sercos_State.S7_FaultReactionActive;
	RETURN;
END_IF

IF NOT stControl.b15_Enable THEN 
	_eState := E_Sercos_State.S3_ReadyToSwitchOn;
	RETURN;
END_IF

IF NOT stControl.b14_Start THEN
	_eState := E_Sercos_State.S6_QuickStop;
	RETURN;
END_IF

IF stControl.b13_Halt THEN
	_eState := E_Sercos_State.S5b_Halt;
	RETURN;
END_IF
END_METHOD

METHOD PRIVATE S5b_Halt : BOOL
VAR_INPUT
END_VAR
stStatus.b15_ReadyToOperate 		:= TRUE;
stStatus.b14_ReadyToOperate 		:= TRUE;
stStatus.b13_Error 					:= FALSE;
stStatus.b7_QuickStop 				:= FALSE;
stStatus.b4_Halt 					:= TRUE;
stStatus.b3_CommandProcessing 		:= FALSE;

IF NOT bPower THEN
	_eState := E_Sercos_State.S2_SwitchOnDisabled;
	RETURN;
END_IF

IF _bError THEN
	_eState := E_Sercos_State.S7_FaultReactionActive;
	RETURN;
END_IF

IF NOT stControl.b15_Enable THEN 
	_eState := E_Sercos_State.S3_ReadyToSwitchOn;
	RETURN;
END_IF

IF NOT stControl.b14_Start THEN
	_eState := E_Sercos_State.S6_QuickStop;
	RETURN;
END_IF

IF NOT stControl.b13_Halt THEN
	_eState := E_Sercos_State.S5a_DriveInOperation;
	RETURN;
END_IF
END_METHOD

METHOD PRIVATE S6_QuickStop : BOOL
VAR_INPUT
END_VAR
stStatus.b15_ReadyToOperate 		:= TRUE;
stStatus.b14_ReadyToOperate 		:= TRUE;
stStatus.b13_Error 					:= FALSE;
stStatus.b7_QuickStop 				:= TRUE;
stStatus.b4_Halt 					:= TRUE;
stStatus.b3_CommandProcessing 		:= FALSE;

IF NOT bPower THEN
	_eState := E_Sercos_State.S2_SwitchOnDisabled;
	RETURN;
END_IF

IF _bError THEN
	_eState := E_Sercos_State.S7_FaultReactionActive;
	RETURN;
END_IF

IF NOT stControl.b15_Enable THEN 
	_eState := E_Sercos_State.S3_ReadyToSwitchOn;
	RETURN;
END_IF

IF stControl.b13_Halt AND stControl.b14_Start THEN
	_eState := E_Sercos_State.S5b_Halt;
	RETURN;
END_IF

IF NOT stControl.b13_Halt AND stControl.b14_Start THEN
	_eState := E_Sercos_State.S5a_DriveInOperation;
	RETURN;
END_IF
END_METHOD

METHOD PRIVATE S7_FaultReactionActive : BOOL
VAR_INPUT
END_VAR
stStatus.b15_ReadyToOperate 		:= TRUE;
stStatus.b14_ReadyToOperate 		:= TRUE;
stStatus.b13_Error 					:= TRUE;
stStatus.b7_QuickStop 				:= FALSE;
stStatus.b4_Halt 					:= FALSE;
stStatus.b3_CommandProcessing 		:= FALSE;

IF NOT bPower THEN
	_eState := E_Sercos_State.S2_SwitchOnDisabled;
	RETURN;
END_IF

_eState := E_Sercos_State.S8_Fault;
END_METHOD

METHOD PRIVATE S8_Fault : BOOL
VAR_INPUT
END_VAR
stStatus.b15_ReadyToOperate 		:= TRUE;
stStatus.b14_ReadyToOperate 		:= FALSE;
stStatus.b13_Error 					:= TRUE;
stStatus.b7_QuickStop 				:= FALSE;
stStatus.b4_Halt 					:= FALSE;
stStatus.b3_CommandProcessing 		:= FALSE;

IF _rTrig_Reset.Q THEN
	_eState := E_Sercos_State.S2_SwitchOnDisabled;
	_bError := FALSE;
	RETURN;	
END_IF
END_METHOD

END_FUNCTION_BLOCK

// Devices/Drives/Sercos/FB_Sercos_VC
(*
	Sercos Velocity Control
	MDT: S-0-0134 Master control word
	MDT: S-0-0036 Velocity command value
	AT: S-0-0135 Drive Status word
	AT: S-0-0051 Position feedback 1 value
*)

{attribute 'reflection'} 
FUNCTION_BLOCK FB_Sercos_VC EXTENDS FB_LinkDataReal 
VAR_INPUT
	pControl			: PVOID; //Pocess data from fieldbus, 4 BYTES FROM FIELDBUS
	pStatus				: PVOID; //Pocess data to fieldbus, 4 BYTES FROM FIELDBUS		
	stControl	 		: ST_Sercos_VC_Control;
	stConfig			: ST_Sercos_VC_Config;
	bSTO 				: BOOL := TRUE;
END_VAR

VAR_OUTPUT
	stStatus 			: ST_Sercos_VC_Status;	
END_VAR

VAR		
	{attribute 'instance-path'} 
    {attribute 'noinit'} 
    _sPath 				: STRING;
	_fbStateMachine 	: FB_Sercos_FSM;
	_fbEncoder 			: FB_Encoder;	
	_fVelocity			: REAL;
END_VAR

SUPER^();
InitRun();

GetControlData();
Cycle();
SetStatusData();

METHOD PRIVATE Cycle
VAR
	fTargetVelocitySign : REAL;
	fTargetVelocityFactor : REAL;
	fTargetVelocity : REAL;	
END_VAR
_fbStateMachine.bPower := bSTO;

_fbStateMachine.stControl := stControl.nControlWord;
_fbStateMachine();
stStatus.nStatusWord := _fbStateMachine.stStatus;

IF (_fbStateMachine._eState = E_Sercos_State.S5a_DriveInOperation OR _fbStateMachine._eState = E_Sercos_State.S5b_Halt) THEN	
	_fbEncoder.fValue := _fVelocity := GetTargetVelocity(stControl.nVelocityCommand, stConfig.fReferenceVelocity, stConfig.fNormalizationFactor);	
	_fbEncoder();
END_IF

stStatus.nStatusWord.b8_Reserved := stControl.nControlWord.b8_Reserved;
stStatus.nStatusWord.b9_Reserved := stControl.nControlWord.b9_Reserved;
stStatus.nStatusWord.b10_OperationMode := stControl.nControlWord.b11_Reserved;

stStatus.nPositionFeedback := _fbEncoder.nResult;

//Set Link Data
IF stConfig.bIsLinkOutputVelocity THEN
	ControlData := LREAL_TO_REAL(_fVelocity);
ELSE
	ControlData := LREAL_TO_REAL(_fbEncoder.fResult);
END_IF
END_METHOD

PROPERTY eState : E_Sercos_State
GET
eState := _fbStateMachine.eState;
END_GET
END_PROPERTY

PROPERTY PUBLIC fbEncoder : REFERENCE TO FB_Encoder
GET
fbEncoder REF= _fbEncoder;
END_GET
END_PROPERTY

METHOD INTERNAL GetControlData
IF pControl <= 0 OR stConfig.bForceMode THEN RETURN; END_IF

(*Control Word*)
F_Memcpy(ADR(stControl), pControl, 2, stConfig.bSwapProcessData);
(*Velocity Command*)
F_Memcpy(ADR(stControl) + 2, pControl + 2, 4, stConfig.bSwapProcessData);
END_METHOD

METHOD INTERNAL GetTargetVelocity : REAL
VAR_INPUT
	nVelocityCommand 			: DINT;
	fReferenceVelocity			: REAL;
	nNormalizationFactor 		: REAL;
END_VAR

VAR
	fTargetVelocity 			: REAL;	
	fTargetVelocitySign 		: REAL;
	fTargetVelocityFactor 		: REAL;	
END_VAR
fTargetVelocity := DINT_TO_REAL(nVelocityCommand);
fTargetVelocityFactor := F_Norm(0, nNormalizationFactor, ABS(fTargetVelocity));
GetTargetVelocity := fReferenceVelocity * fTargetVelocityFactor * F_Sign(fTargetVelocity);
END_METHOD

METHOD PRIVATE InitRun
VAR_INST
	bInitRun : BOOL := TRUE;
END_VAR
IF NOT bInitRun THEN RETURN; END_IF
bInitRun := FALSE;

IF pControl = 0 OR pStatus = 0 THEN
	ADSLOGSTR(ADSLOG_MSGTYPE_WARN, '%s', CONCAT(_sPath, ' PLC IO is not assigned!'));	
END_IF

_fbEncoder.stConfig.bIsIntegrator := TRUE;
END_METHOD

METHOD PRIVATE Motion : REAL
VAR_INPUT
END_VAR
END_METHOD

METHOD INTERNAL SetStatusData
IF pStatus <= 0 THEN RETURN; END_IF

(*StatusWord*)
F_Memcpy(pStatus, ADR(stStatus), 2, stConfig.bSwapProcessData);
(*Position Feedback*)
F_Memcpy(pStatus + 2, ADR(stStatus) + 2, 4, stConfig.bSwapProcessData);
END_METHOD

END_FUNCTION_BLOCK

// Devices/Terminals/FB_Beckhoff_EL6001/FB_Beckhoff_EL6001
FUNCTION_BLOCK FB_Beckhoff_EL6001
VAR_INPUT
	bSend				: BOOL;
	nLength				: UINT;
	pDataIn				: POINTER TO BYTE; //Data to send
	pDataOut			: POINTER TO BYTE; //Received data when nDataAvailable > 0.
END_VAR

VAR_OUTPUT
	bBusy				: BOOL;
	nDataAvailable		: INT; //Received bytes. Only available for one cycle.
END_VAR

VAR
	nControl			AT %I* : UINT;
	nDataOut			AT %I* : ARRAY[0..21] OF USINT;
	nStatus				AT %Q* : UINT;
	nDataIn				AT %Q* : ARRAY[0..21] OF USINT;
END_VAR

VAR
	_nControlByte			: BYTE;
	_nOutLength				: BYTE;	
	_bTransmitRequest		: BOOL;
	_bReceiveAccecpted		: BOOL;
	_bInitRequest			: BOOL;
	_bSendContinuous		: BOOL;
	
	_bTransmitAccepted		: BOOL;
	_bReceiveRequest		: BOOL;
	_bInitAccepted			: BOOL;
	_bBufferFull			: BOOL;
	_bParityError			: BOOL;
	_bFramingError			: BOOL;
	_bOverrunError			: BOOL;
	_nInLength				: BYTE;
	
	_nPendingLength			: UINT;
	_nOffsetNext			: UINT;
	
	_eState					: E_Beckhoff_EL6001_State;
	_trigSend				: R_TRIG;
END_VAR

(* Receive control word *)
	_bTransmitRequest 	:= nControl.0 <> _nControlByte.0;
	_bReceiveAccecpted 	:= nControl.1 <> _nControlByte.1;
	_bInitRequest		:= nControl = 4;
	_bSendContinuous		:= nControl.3 AND NOT _nControlByte.0;	
	_nControlByte 		:= F_GetLByte(nControl);
	_nOutLength 			:= F_GetHByte(nControl);

(* Initialize *)
	IF _bInitRequest THEN
		_eState := E_Beckhoff_EL6001_State.INIT;			
	END_IF
	
CASE _eState OF
	E_Beckhoff_EL6001_State.INIT:
		_bTransmitAccepted 	:= FALSE;
		_bReceiveRequest		:= FALSE;
		_bInitAccepted		:= TRUE;
		_bBufferFull			:= FALSE;
		_bParityError		:= FALSE;
		_bFramingError		:= FALSE;
		_bOverrunError		:= FALSE;
		_nInLength			:= 0;
		nDataAvailable		:= 0;
		
		// -> INIT_READY
		IF nControl = 0 THEN
			_bInitAccepted := FALSE;		
			_eState := E_Beckhoff_EL6001_State.READY;
		END_IF

	E_Beckhoff_EL6001_State.READY:
		nDataAvailable := 0;

		// -> TRANSMIT
		IF _bTransmitRequest AND _nOutLength > 0 AND _nOutLength < 23 THEN
			_eState := E_Beckhoff_EL6001_State.TRANSMIT;
			RETURN;
		END_IF
		
		_trigSend(CLK := bSend);
		
		// -> RECEIVE
		IF _trigSend.Q AND nLength > 0 AND pDataIn <> 0 THEN
			_bReceiveRequest := NOT _bReceiveRequest;
			_nPendingLength := nLength;
			_nInLength := UINT_TO_BYTE(MIN(22, _nPendingLength));
			memcpy(ADR(nDataIn), pDataIn, _nInLength);		
			_eState := E_Beckhoff_EL6001_State.RECEIVE;
		END_IF	
		
	E_Beckhoff_EL6001_State.TRANSMIT:
		IF pDataOut <> 0 THEN
			memcpy(pDataOut, ADR(nDataOut), _nOutLength);
		END_IF
		_bTransmitAccepted := NOT _bTransmitAccepted;
		nDataAvailable := _nOutLength;
		_eState := E_Beckhoff_EL6001_State.READY;
		
	E_Beckhoff_EL6001_State.RECEIVE:
		IF _bReceiveAccecpted THEN
			_nOffsetNext := _nInLength;
			_nPendingLength := _nPendingLength - _nOffsetNext;
			IF _nPendingLength = 0 THEN
				_eState := E_Beckhoff_EL6001_State.READY;
			END_IF
			IF _nPendingLength > 0 THEN
				_bReceiveRequest := NOT _bReceiveRequest;
				_nInLength := UINT_TO_BYTE(MIN(22, _nPendingLength));
				memcpy(ADR(nDataIn), pDataIn + _nOffsetNext, _nInLength);
				_eState := E_Beckhoff_EL6001_State.RECEIVE;
			END_IF				
		END_IF
	
END_CASE

bBusy := _eState <> E_Beckhoff_EL6001_State.READY;
	
(* Send status word *)
	nStatus.0			:= _bTransmitAccepted;
	nStatus.1			:= _bReceiveRequest;
	nStatus.2			:= _bInitAccepted;
	nStatus.3			:= _bBufferFull;
	nStatus.4			:= _bParityError;
	nStatus.5			:= _bFramingError;
	nStatus.6			:= _bOverrunError;
	memcpy(ADR(nStatus) + 1, ADR(_nInLength), 1);

PROPERTY INTERNAL BufferFull : BOOl
GET
BufferFull := _bBufferFull;
END_GET
END_PROPERTY

PROPERTY INTERNAL Control : UINT
SET
nControl := Control;
END_SET
END_PROPERTY

PROPERTY INTERNAL FramingError : BOOl
GET
FramingError := _bFramingError;
END_GET
END_PROPERTY

PROPERTY INTERNAL InitAccepted : BOOl
GET
InitAccepted := _bInitAccepted;
END_GET
END_PROPERTY

PROPERTY INTERNAL InitRequest : BOOl
GET
InitRequest := _bInitRequest;
END_GET
END_PROPERTY

PROPERTY INTERNAL OverrunError : BOOl
GET
OverrunError := _bOverrunError;
END_GET
END_PROPERTY

PROPERTY INTERNAL ParityError : BOOl
GET
ParityError := _bParityError;
END_GET
END_PROPERTY

PROPERTY INTERNAL ReceiveAccepted : BOOl
GET
ReceiveAccepted := _bReceiveAccecpted;
END_GET
END_PROPERTY

PROPERTY INTERNAL ReceiveRequest : BOOl
GET
ReceiveRequest := _bReceiveRequest;
END_GET
END_PROPERTY

PROPERTY INTERNAL SendContinuous : BOOl
GET
SendContinuous := _bSendContinuous;
END_GET
END_PROPERTY

PROPERTY INTERNAL State : E_Beckhoff_EL6001_State
GET
State := _eState;
END_GET
SET
_eState := State;
END_SET
END_PROPERTY

PROPERTY INTERNAL TransmitAccepted : BOOl
GET
TransmitAccepted := _bTransmitAccepted;
END_GET
END_PROPERTY

PROPERTY INTERNAL TransmitRequest : BOOl
GET
TransmitRequest := _bTransmitRequest;
END_GET
END_PROPERTY

END_FUNCTION_BLOCK

// Devices/Terminals/FB_Beckhoff_EJ1918
FUNCTION_BLOCK FB_Beckhoff_EJ1918
VAR_INPUT
	bIn1			: BOOL;
	bIn2			: BOOL;
	bIn3			: BOOL;
	bIn4			: BOOL;
END_VAR
VAR
	RxPDO			AT %I* : FSOE_6;
	TxPDO			AT %Q* : FSOE_7;	
	fbFsoeSlave		: FB_FsoeSlave;
	nMasterData		: BYTE := 0;
	nSlaveData		: WORD := 0;
END_VAR

nSlaveData.0 := bIn1;
nSlaveData.1 := bIn1;
nSlaveData.3 := bIn2;
nSlaveData.4 := bIn2;
nSlaveData.6 := bIn3;
nSlaveData.7 := bIn3;
nSlaveData.9 := bIn4;
nSlaveData.10 := bIn4;

fbFsoeSlave();

METHOD FB_init : BOOL
VAR_INPUT
	bInitRetains 	: BOOL; // if TRUE, the retain variables are initialized (warm start / cold start)
	bInCopyCode 	: BOOL;  // if TRUE, the instance afterwards gets moved into the copy code (online change)
END_VAR
fbFsoeSlave.stConfig.nSlaveAddress := 0;
fbFsoeSlave.stConfig.pFromBus := ADR(RxPDO);
fbFsoeSlave.stConfig.pToBus := ADR(TxPDO);
fbFsoeSlave.stConfig.nSizeMaster := 6;
fbFsoeSlave.stConfig.nSizeSlave := 7;
fbFsoeSlave.stConfig.pMasterData := ADR(nMasterData);
fbFsoeSlave.stConfig.pSlaveData := ADR(nSlaveData);
END_METHOD

END_FUNCTION_BLOCK

// Devices/Terminals/FB_Beckhoff_EK1914
FUNCTION_BLOCK FB_Beckhoff_EK1914
VAR_INPUT
	bSafetyIn1		: BOOL;
	bSafetyIn2		: BOOL;
	bInput0			: BOOL;
	bInput1			: BOOL;
	bInput2			: BOOL;
	bInput3			: BOOL;
END_VAR
VAR_OUTPUT
	bSafetyOut1		: BOOL;
	bSafetyOut2		: BOOL;
	bOutput0		: BOOL;
	bOutput1		: BOOL;
	bOutput2		: BOOL;
	bOutput3		: BOOL;
	bOSafetyLinkedOutput0 : BOOL;
	bOSafetyLinkedOutput1 : BOOL;
END_VAR
VAR
	RxPDO			AT %I* : FSOE_6;
	TxPDO			AT %Q* : FSOE_6;	
	fbFsoeSlave		: FB_FsoeSlave;
	nMasterData		: BYTE := 0;
	nSlaveData		: BYTE := 0;
	
	bOutputDIO0		AT %I* : BOOL;
	bOutputDIO1		AT %I* : BOOL;
	bOutputDIO2		AT %I* : BOOL;
	bOutputDIO3		AT %I* : BOOL;
	bOutputDIOSafetyLinkedOutput0		AT %I* : BOOL;
	bOutputDIOSafetyLinkedOutput1		AT %I* : BOOL;
	bInputDIO0		AT %Q* : BOOL;
	bInputDIO1		AT %Q* : BOOL;
	bInputDIO2		AT %Q* : BOOL;
	bInputDIO3		AT %Q* : BOOL;
END_VAR

nSlaveData.0 := bSafetyIn1;
nSlaveData.1 := bSafetyIn2;
bInputDIO0 := bInput0;
bInputDIO1 := bInput1;
bInputDIO2 := bInput2;
bInputDIO3 := bInput3;

fbFsoeSlave();

bSafetyOut1 := nMasterData.0;
bSafetyOut2 := nMasterData.1;
bOutput0 := bOutputDIO0;
bOutput1 := bOutputDIO1;
bOutput2 := bOutputDIO2;
bOutput3 := bOutputDIO3;
bOSafetyLinkedOutput0 := bOutputDIOSafetyLinkedOutput0;
bOSafetyLinkedOutput1 := bOutputDIOSafetyLinkedOutput1;

METHOD FB_init : BOOL
VAR_INPUT
	bInitRetains 	: BOOL; // if TRUE, the retain variables are initialized (warm start / cold start)
	bInCopyCode 	: BOOL;  // if TRUE, the instance afterwards gets moved into the copy code (online change)
END_VAR
fbFsoeSlave.stConfig.nSlaveAddress := 0;
fbFsoeSlave.stConfig.pFromBus := ADR(RxPDO);
fbFsoeSlave.stConfig.pToBus := ADR(TxPDO);
fbFsoeSlave.stConfig.nSizeMaster := 6;
fbFsoeSlave.stConfig.nSizeSlave := 6;
fbFsoeSlave.stConfig.pMasterData := ADR(nMasterData);
fbFsoeSlave.stConfig.pSlaveData := ADR(nSlaveData);
END_METHOD

END_FUNCTION_BLOCK

// Devices/Terminals/FB_Beckhoff_EL1904
FUNCTION_BLOCK FB_Beckhoff_EL1904
VAR_INPUT
	bIn1			: BOOL;
	bIn2			: BOOL;
	bIn3			: BOOL;
	bIn4			: BOOL;
END_VAR
VAR
	RxPDO			AT %I* : FSOE_6;
	TxPDO			AT %Q* : FSOE_6;	
	fbFsoeSlave		: FB_FsoeSlave;
	nMasterData		: BYTE := 0;
	nSlaveData		: BYTE := 0;
END_VAR

nSlaveData.0 := bIn1;
nSlaveData.1 := bIn2;
nSlaveData.2 := bIn3;
nSlaveData.3 := bIn4;

fbFsoeSlave();

METHOD FB_init : BOOL
VAR_INPUT
	bInitRetains 	: BOOL; // if TRUE, the retain variables are initialized (warm start / cold start)
	bInCopyCode 	: BOOL;  // if TRUE, the instance afterwards gets moved into the copy code (online change)
END_VAR
fbFsoeSlave.stConfig.nSlaveAddress := 0;
fbFsoeSlave.stConfig.pFromBus := ADR(RxPDO);
fbFsoeSlave.stConfig.pToBus := ADR(TxPDO);
fbFsoeSlave.stConfig.nSizeMaster := 6;
fbFsoeSlave.stConfig.nSizeSlave := 6;
fbFsoeSlave.stConfig.pMasterData := ADR(nMasterData);
fbFsoeSlave.stConfig.pSlaveData := ADR(nSlaveData);
END_METHOD

END_FUNCTION_BLOCK

// Devices/Terminals/FB_Beckhoff_EL1918
FUNCTION_BLOCK FB_Beckhoff_EL1918
VAR_INPUT
	bIn1			: BOOL;
	bIn2			: BOOL;
	bIn3			: BOOL;
	bIn4			: BOOL;
	bIn5			: BOOL;
	bIn6			: BOOL;
	bIn7			: BOOL;
	bIn8			: BOOL;
END_VAR
VAR
	RxPDO			AT %I* : FSOE_6;
	TxPDO			AT %Q* : FSOE_7;	
	fbFsoeSlave		: FB_FsoeSlave;
	nMasterData		: BYTE := 0;
	nSlaveData		: WORD := 0;
END_VAR

nSlaveData.0 := bIn1;
nSlaveData.2 := bIn2;
nSlaveData.4 := bIn3;
nSlaveData.6 := bIn4;
nSlaveData.8 := bIn5;
nSlaveData.10 := bIn6;
nSlaveData.12 := bIn7;
nSlaveData.14 := bIn8;

fbFsoeSlave();

METHOD FB_init : BOOL
VAR_INPUT
	bInitRetains 	: BOOL; // if TRUE, the retain variables are initialized (warm start / cold start)
	bInCopyCode 	: BOOL;  // if TRUE, the instance afterwards gets moved into the copy code (online change)
END_VAR
fbFsoeSlave.stConfig.nSlaveAddress := 0;
fbFsoeSlave.stConfig.pFromBus := ADR(RxPDO);
fbFsoeSlave.stConfig.pToBus := ADR(TxPDO);
fbFsoeSlave.stConfig.nSizeMaster := 6;
fbFsoeSlave.stConfig.nSizeSlave := 7;
fbFsoeSlave.stConfig.pMasterData := ADR(nMasterData);
fbFsoeSlave.stConfig.pSlaveData := ADR(nSlaveData);
END_METHOD

END_FUNCTION_BLOCK

// Devices/Terminals/FB_Beckhoff_EL2904
FUNCTION_BLOCK FB_Beckhoff_EL2904
VAR_OUTPUT
	bOut1			: BOOL;
	bOut2			: BOOL;
	bOut3			: BOOL;
	bOut4			: BOOL;	
END_VAR
VAR
	RxPDO			AT %I* : FSOE_6;
	TxPDO			AT %Q* : FSOE_6;	
	fbFsoeSlave		: FB_FsoeSlave;
	nMasterData		: BYTE := 0;
	nSlaveData		: BYTE := 0;
END_VAR

fbFsoeSlave();

bOut1 := nMasterData.0;
bOut2 := nMasterData.1;
bOut3 := nMasterData.2;
bOut4 := nMasterData.3;

METHOD FB_init : BOOL
VAR_INPUT
	bInitRetains 	: BOOL; // if TRUE, the retain variables are initialized (warm start / cold start)
	bInCopyCode 	: BOOL;  // if TRUE, the instance afterwards gets moved into the copy code (online change)
END_VAR
fbFsoeSlave.stConfig.nSlaveAddress := 0;
fbFsoeSlave.stConfig.pFromBus := ADR(RxPDO);
fbFsoeSlave.stConfig.pToBus := ADR(TxPDO);
fbFsoeSlave.stConfig.nSizeMaster := 6;
fbFsoeSlave.stConfig.nSizeSlave := 6;
fbFsoeSlave.stConfig.pMasterData := ADR(nMasterData);
fbFsoeSlave.stConfig.pSlaveData := ADR(nSlaveData);
END_METHOD

END_FUNCTION_BLOCK

// Devices/Terminals/FB_Beckhoff_EL5152
FUNCTION_BLOCK FB_Beckhoff_EL5152
VAR_INPUT
	nValue1		: UINT;
	nValue2		: UINT;
END_VAR
VAR
	nControl1		AT %I* : UINT;
	nSetCounter1	AT %I* : UINT;
	nControl2		AT %I* : UINT;
	nSetCounter2	AT %I* : UINT;
	
	nStatus1		AT %Q* : UINT;
	nCounter1		AT %Q* : UINT;	
	nPeriod1    	AT %Q* : UDINT;
	nStatus2		AT %Q* : UINT;
	nCounter2		AT %Q* : UINT;
	nPeriod2    	AT %Q* : UDINT;
END_VAR

nStatus1.2 := nControl1.2;
nStatus2.2 := nControl2.2;

nCounter1 := nValue1;
nCounter2 := nValue2;

PROPERTY INTERNAL Control1 : UINT
SET
nControl1 := Control1;
END_SET
END_PROPERTY

PROPERTY INTERNAL Control2 : UINT
SET
nControl2 := Control2;
END_SET
END_PROPERTY

PROPERTY INTERNAL Counter1 : UINT
GET
Counter1 := nCounter1;
END_GET
END_PROPERTY

PROPERTY INTERNAL Counter2 : UINT
GET
Counter2 := nCounter2;
END_GET
END_PROPERTY

PROPERTY INTERNAL Period1 : UDINT
GET
Period1 := nPeriod1;
END_GET
END_PROPERTY

PROPERTY INTERNAL Period2 : UDINT
GET
Period2 := nPeriod2;
END_GET
END_PROPERTY

PROPERTY INTERNAL SetCounter1 : UINT
SET
nSetCounter1 := SetCounter1;
END_SET
END_PROPERTY

PROPERTY INTERNAL SetCounter2 : UINT
SET
nSetCounter2 := SetCounter2;
END_SET
END_PROPERTY

PROPERTY INTERNAL Status1 : UINT
GET
Status1 := nStatus1;
END_GET
END_PROPERTY

PROPERTY INTERNAL Status2 : UINT
GET
Status2 := nStatus2;
END_GET
END_PROPERTY

END_FUNCTION_BLOCK

// Devices/Terminals/FB_FSOE_19
FUNCTION_BLOCK FB_FSOE_19
VAR_INPUT
	SafetyIn				: ULINT;
END_VAR
VAR_OUTPUT
	SafetyOut				: ULINT;
END_VAR
VAR
	RxPDO			AT %I* 	: FSOE_19;
	TxPDO			AT %Q* 	: FSOE_19;
	fbFsoeSlave				: FB_FsoeSlave;
END_VAR

fbFsoeSlave();

METHOD FB_init : BOOL
VAR_INPUT
	bInitRetains : BOOL; // if TRUE, the retain variables are initialized (warm start / cold start)
	bInCopyCode : BOOL;  // if TRUE, the instance afterwards gets moved into the copy code (online change)
END_VAR
fbFsoeSlave.stConfig.nSlaveAddress := 0;
fbFsoeSlave.stConfig.pFromBus := ADR(RxPDO);
fbFsoeSlave.stConfig.pToBus := ADR(TxPDO);
fbFsoeSlave.stConfig.nSizeMaster := 19;
fbFsoeSlave.stConfig.nSizeSlave := 19;
fbFsoeSlave.stConfig.pMasterData := ADR(SafetyOut);
fbFsoeSlave.stConfig.pSlaveData := ADR(SafetyIn);
END_METHOD

END_FUNCTION_BLOCK
